RoboDK station: ChArUco Hand-Eye Calibration - v2.rdk

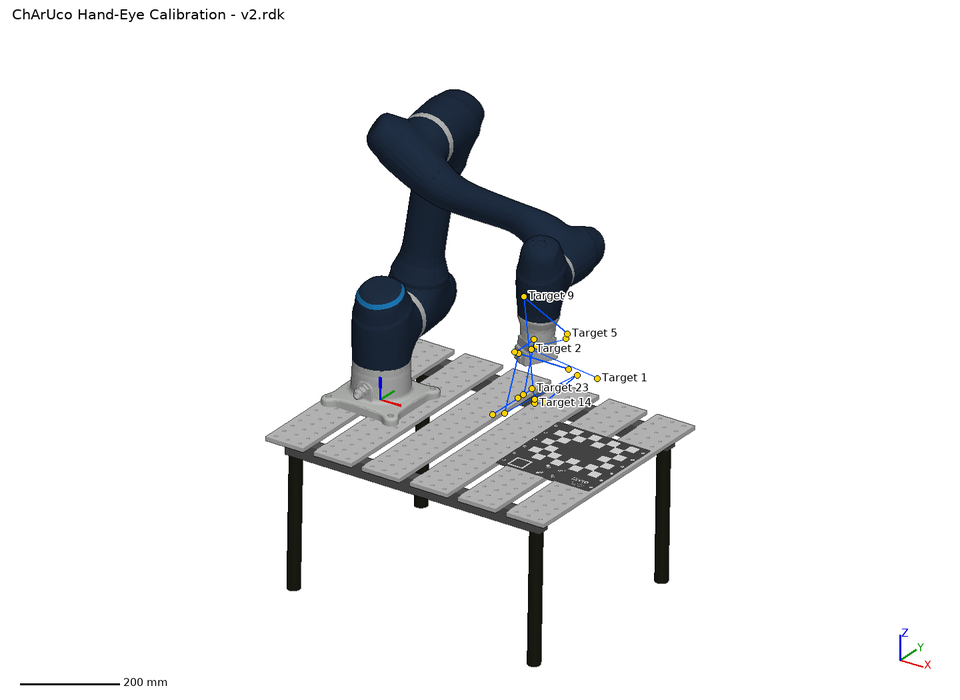
[picture v0: the station drawn from its stored meshes, robots at their saved joint values, targets as dots, program paths as lines]
Station Charuco Test Station (saved by RoboDK 5.9.2). Poses are relative to the parent item; angles as X-Y-Z fixed-axis rotations.
Station parameters (name, value as stored): IO_2, 0, IO_5, 1, IO_3, 0, 2, 0, 3, 0
  - program declamping (2 instructions, listed below)
  - program clamping (2 instructions, listed below)
  - frame World at (231.85, -7.07, -1.69) mm, rotated rx 0 ry -1.78 rz 1.07 deg
    - frame Doosan Robotics A0509 Base at (0, 0, 0) mm, rotated rx 0 ry 2.86 rz 0 deg
      - robot Doosan Robotics A0509: 6 axes, payload 5 kg, reach 900 mm, repeatability 0.03 mm
          modified DH rows (alpha deg, a mm, theta deg, d mm): 0, 0, 0, 155.5; -90, 0, -90, 0; 0, 409, -90, 0; -90, 0, 0, 367; 90, 0, 0, 0; -90, 0, 90, 124
          base shift (0, 0, 0) mm, rotated rx 0 ry 0 rz 180 deg
          joint limits [-360, -360, -150, -360, -360, -360] to [360, 360, 150, 360, 360, 360]; home [0, 0, 90, 0, 0, 0]; saved at [6.063, 7.68, 117.075, 0.353, 58.096, 120.775]
        - tool 560210_HGPT-35-A-B, TCP at (80, 0, 45) mm, size 42 x 50.8 x 80 mm, geometry from World
    - target Target 1 (Cartesian target) at (529.19, 0, 173.22) mm, rotated rx -180 ry 0 rz 0 deg; joints [0, 12.117, 98.841, 0, 66.184, 180] of Doosan Robotics A0509
    - target Target 2 (Cartesian target) at (349.42, 30.06, 182.74) mm, rotated rx -178.17 ry -2.18 rz 139.97 deg; joints [5.054, 0.015, 111.663, 0, 68.31, 45.053] of Doosan Robotics A0509
    - target Target 3 (Cartesian target) at (349.4, 50.08, 182.68) mm, rotated rx -177.24 ry -0.74 rz 105.07 deg; joints [8.384, 0.348, 111.339, 0, 68.311, 83.296] of Doosan Robotics A0509
    - target Target 4 (Cartesian target) at (379.39, 110.18, 181.14) mm, rotated rx -177.4 ry 1.21 rz 65.12 deg; joints [16.587, 6.181, 105.115, 0, 68.712, 131.494] of Doosan Robotics A0509
    - target Target 5 (Cartesian target) at (369.32, 130.03, 181.73) mm, rotated rx 180 ry 7.15 rz 179.99 deg; joints [22.111, 0.807, 111.453, -4.393, 58.532, 24.108] of Doosan Robotics A0509
    - target Target 6 (Cartesian target) at (369.31, 130.01, 181.73) mm, rotated rx 175.39 ry 5.47 rz 139.77 deg; joints [22.109, 0.806, 111.455, -4.394, 58.531, 64.112] of Doosan Robotics A0509
    - target Target 7 (Cartesian target) at (369.32, 130.02, 181.73) mm, rotated rx 172.96 ry 1.23 rz 99.91 deg; joints [22.111, 0.806, 111.453, -4.394, 58.531, 104.117] of Doosan Robotics A0509
    - target Target 8 (Cartesian target) at (369.32, 130.02, 181.73) mm, rotated rx 173.8 ry -3.57 rz 60.18 deg; joints [22.11, 0.806, 111.454, -4.394, 58.532, 144.118] of Doosan Robotics A0509
    - target Target 9 (Cartesian target) at (355.87, -0.03, 312.67) mm, rotated rx 180 ry -2.84 rz 180 deg; joints [-0.007, -3.813, 94.527, 0.002, 89.271, -0.002] of Doosan Robotics A0509
    - target Target 11 (Cartesian target) at (355.87, -0.03, 312.67) mm, rotated rx -178.17 ry -2.18 rz 139.96 deg; joints [-0.007, -3.813, 94.527, 0.002, 89.271, 40.001] of Doosan Robotics A0509
    - target Target 12 (Cartesian target) at (355.87, -0.03, 312.67) mm, rotated rx -177.16 ry 0 rz 89.99 deg; joints [-0.007, -3.813, 94.527, 0.002, 89.271, 90.002] of Doosan Robotics A0509
    - target Target 13 (Cartesian target) at (355.87, -0.03, 312.67) mm, rotated rx 177.82 ry -1.83 rz -129.97 deg; joints [-0.007, -3.813, 94.527, 0.002, 89.271, -50.005] of Doosan Robotics A0509
    - target Target 14 (Cartesian target) at (374.31, -0.04, 81.5) mm, rotated rx 180 ry -2.85 rz -180 deg; joints [-0.006, 11.5, 116.754, 0, 51.737, -0.008] of Doosan Robotics A0509
    - target Target 15 (Cartesian target) at (400.01, 0.06, 90.18) mm, rotated rx -174.02 ry -10.47 rz -170.32 deg; joints [4.153, 17.227, 107.795, -8.099, 62.218, -1.647] of Doosan Robotics A0509
    - target Target 16 (Cartesian target) at (390.18, 130.07, 95.59) mm, rotated rx -161.09 ry 7.32 rz 151.77 deg; joints [28.44, 19.616, 105.419, -19.231, 66.069, 67.975] of Doosan Robotics A0509
    - target Target 17 (Cartesian target) at (390.99, -130.12, 115.57) mm, rotated rx -175.43 ry 6.23 rz -99.85 deg; joints [-23.319, 10.299, 112.249, 10.436, 52.261, -109.378] of Doosan Robotics A0509
    - target Target 18 (Cartesian target) at (339.55, 0.01, 183.15) mm, rotated rx 180 ry -2.86 rz -180 deg; joints [0.001, -1.553, 113.219, 0, 68.333, 0.001] of Doosan Robotics A0509
    - target Target 19 (Cartesian target) at (459.59, 0, 177.15) mm, rotated rx -180 ry -32.86 rz 180 deg; joints [0, 31.451, 75.378, 0.001, 103.173, 0.001] of Doosan Robotics A0509
    - target Target 20 (Cartesian target) at (329.62, 0, 183.64) mm, rotated rx 180 ry 17.14 rz 180 deg; joints [0.001, -13.948, 125.935, -0.001, 48.012, 0.004] of Doosan Robotics A0509
    - target Target 21 (Cartesian target) at (329.63, 70.09, 183.68) mm, rotated rx 166.99 ry 11.34 rz 118.8 deg; joints [19.01, -11.541, 124.161, -12.435, 50.393, 85.516] of Doosan Robotics A0509
    - target Target 22 (Cartesian target) at (427.42, -114.48, 159.86) mm, rotated rx 159.85 ry -25.39 rz 175.54 deg; joints [-22.037, 28.204, 83.669, 12.941, 95.356, -15.486] of Doosan Robotics A0509
    - target Target 23 (Cartesian target) at (427.42, -84.44, 159.8) mm, rotated rx -171.39 ry -30.94 rz 118.56 deg; joints [-18.987, 26.841, 85.802, 14.306, 93.951, 37.089] of Doosan Robotics A0509
    - target Target 24 (Cartesian target) at (427.43, -134.49, 159.8) mm, rotated rx 149 ry 8.39 rz -121.38 deg; joints [-23.999, 29.24, 82.048, 12.052, 96.33, -87.146] of Doosan Robotics A0509
    - target Target 25 (Cartesian target) at (427.45, -224.66, 159.79) mm, rotated rx 176.37 ry 39.55 rz -100.8 deg; joints [-42.998, 30.663, 83.645, 32.018, 90.964, -131.346] of Doosan Robotics A0509
    - object Table 1200x1000mm (Welding) at (239.71, 0, -11.96) mm, rotated rx 0 ry 2.86 rz 0 deg, size 671.5 x 542.9 x 342.9 mm, geometry from Table-1200x1000mm-Welding.sld
      - object Zivid ZVDA-CB01 Calibration Board at (103.57, -98.2, 0.2) mm, size 225 x 225 x 1.5 mm, geometry from Zivid-ZVDA-CB01-Calibration-Board.sld
    - target Detection Zone (Cartesian target) at (374.43, -0.02, 90.12) mm, rotated rx 180 ry -2.65 rz 179.96 deg; joints [-0.007, 10.783, 116.197, 0.008, 52.992, 0.024] of Doosan Robotics A0509
  - program Prog3 (49 instructions, listed below)
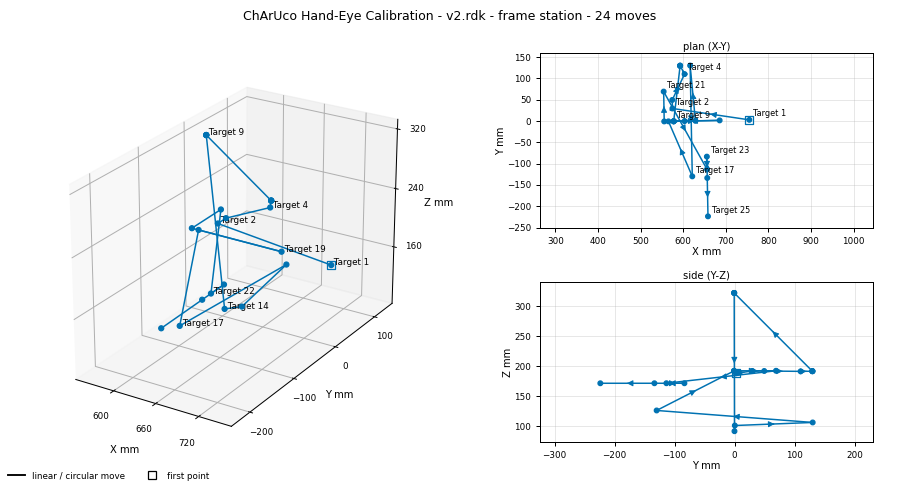
[picture p0: tool path of ChArUco Hand-Eye Calibration - v2.rdk in frame station, 24 of 24 moves have a stored position in this frame; points joined in program order, loops and branches not executed]

--- program declamping (robot Doosan Robotics A0509) ---
  Set IO_2=1
  Set IO_2=0

--- program clamping (robot Doosan Robotics A0509) ---
  Set IO_3=1
  Set IO_3=0

--- program Prog3 (robot Doosan Robotics A0509) ---
  Set Ref.: World
  Set Tool: 560210_HGPT-35-A-B
  MoveJ (Target 1)
  Pause 2.0 s
  MoveL (Target 2)
  Pause 2.0 s
  MoveL (Target 3)
  Pause 2.0 s
  MoveL (Target 4)
  Pause 2.0 s
  MoveL (Target 5)
  Pause 2.0 s
  MoveL (Target 6)
  Pause 2.0 s
  MoveL (Target 7)
  Pause 2.0 s
  MoveL (Target 8)
  Pause 2.0 s
  MoveL (Target 9)
  Pause 2.0 s
  MoveL (Target 11)
  Pause 2.0 s
  MoveL (Target 12)
  Pause 2.0 s
  MoveL (Target 13)
  Pause 2.0 s
  MoveL (Target 14)
  Pause 2.0 s
  MoveL (Target 15)
  Pause 2.0 s
  MoveL (Target 16)
  Pause 2.0 s
  MoveL (Target 17)
  Pause 2.0 s
  MoveL (Target 18)
  Pause 2.0 s
  MoveL (Target 19)
  Pause 2.0 s
  MoveL (Target 20)
  Pause 2.0 s
  MoveL (Target 21)
  Pause 2.0 s
  MoveL (Target 22)
  Pause 2.0 s
  MoveL (Target 23)
  Pause 2.0 s
  MoveL (Target 24)
  Pause 2.0 s
  MoveL (Target 25)
